(*
    This function block is responsible for printing the results of the assertions using the built-in
    ADSLOGSTR functionality provided by the Tc2_System library. This sends the result using ADS, which
    is consumed by the error list of Visual Studio.
*)
FUNCTION_BLOCK FB_AdsAssertMessageFormatter EXTENDS Base.FB_BaseStatic IMPLEMENTS I_AssertMessageFormatter

METHOD PUBLIC LogAssertFailure
VAR_INPUT
    Expected : T_MaxString;
    Actual : T_MaxString;
    Message : T_MaxString;
    TestInstancePath : T_MaxString;
END_VAR
VAR
    AdjustAssertFailureMessageToMax253CharLength : FB_AdjustAssertFailureMessageToMax253CharLength;
    TestInstancePathCleaned : T_MaxString;
    TestInstancePathFinal : T_MaxString;
    ReturnValue : DINT;
    TestInstancePathProcessed : T_MaxString;
    MessageProcessed : T_MaxString;
    TraceMessage : T_MaxString;
END_VAR
TestInstancePathCleaned := F_RemoveInstancePathAndProjectNameFromTestInstancePath(TestInstancePath);
TestInstancePathFinal := CONCAT(STR1 := 'FAILED TEST $'',
                                STR2 := TestInstancePathCleaned);
TestInstancePathFinal := CONCAT(STR1 := TestInstancePathFinal,
                                STR2 := '$'');

TestInstancePathFinal := CONCAT(STR1 := TestInstancePathFinal,
                                STR2 := ', EXP: ');
TestInstancePathFinal := CONCAT(STR1 := TestInstancePathFinal,
                                STR2 := Expected);
TestInstancePathFinal := CONCAT(STR1 := TestInstancePathFinal,
                                STR2 := ', ACT: ');
TestInstancePathFinal := CONCAT(STR1 := TestInstancePathFinal,
                                STR2 := Actual);
IF LEN(STR := Message) > 0 THEN
    TestInstancePathFinal := CONCAT(STR1 := TestInstancePathFinal,
                                    STR2 := ', MSG: %s');
END_IF

AdjustAssertFailureMessageToMax253CharLength(TestInstancePath := TestInstancePathFinal,
                                             TestMessage := Message,
                                             TestInstancePathProcessed => TestInstancePathProcessed,
                                             TestMessageProcessed => MessageProcessed);

GVL_TcUnit.AdsMessageQueue.WriteLog(MsgCtrlMask := ADSLOG_MSGTYPE_ERROR,
                                    MsgFmtStr := TestInstancePathProcessed,
                                    StrArg := MessageProcessed);

TraceMessage := CONCAT(STR1 := 'ASSERT FAIL $'', STR2 := TestInstancePathCleaned);
TraceMessage := CONCAT(STR1 := TraceMessage, STR2 := '$', EXP: ');
TraceMessage := CONCAT(STR1 := TraceMessage, STR2 := Expected);
TraceMessage := CONCAT(STR1 := TraceMessage, STR2 := ', ACT: ');
TraceMessage := CONCAT(STR1 := TraceMessage, STR2 := Actual);
IF LEN(STR := Message) > 0 THEN
    TraceMessage := CONCAT(STR1 := TraceMessage, STR2 := ', MSG: ');
    TraceMessage := CONCAT(STR1 := TraceMessage, STR2 := Message);
END_IF
TraceWithSeverity(Message := TraceMessage, Severity := Global.TcEventSeverity.Error);
END_METHOD

END_FUNCTION_BLOCK

(* stored: Version 1.1.0.1
   POU FB_AdsAssertMessageFormatter: Id {54911d7d-b4a4-43a8-a981-a2fc14a13f71}, SpecialFunc None
   Method LogAssertFailure: Id {48cbc6b0-5380-44b8-a045-57b6ad9f189d} *)
